{attribute 'GeneratedUsingTerminal: EK1122-0000-0018'}
{attribute addProperty BoxType "EK1122-0000-0018"}
{attribute addProperty Id "Beckhoff_EL15xxsub_EK1100EK1100_1FC0878B2"}
{attribute addProperty CRC "1483514227"}
{attribute addProperty Size "2"}
TYPE Beckhoff_EL15xxEK1122_586CA173 EXTENDS EK1122_1FC0878B :
STRUCT
	{attribute addProperty Name "Beckhoff_EL15xxsub_EK1100"}
	Beckhoff_EL15xxsub_EK1100 : EK1100_1FC0878B;
END_STRUCT
END_TYPE

(* stored: Version 1.2.0.0, ProductVersion 3.1.4024.9
   DUT Beckhoff_EL15xxEK1122_586CA173: Id {a3b4672f-70c9-49ce-ba65-6d981fc89c75} *)
